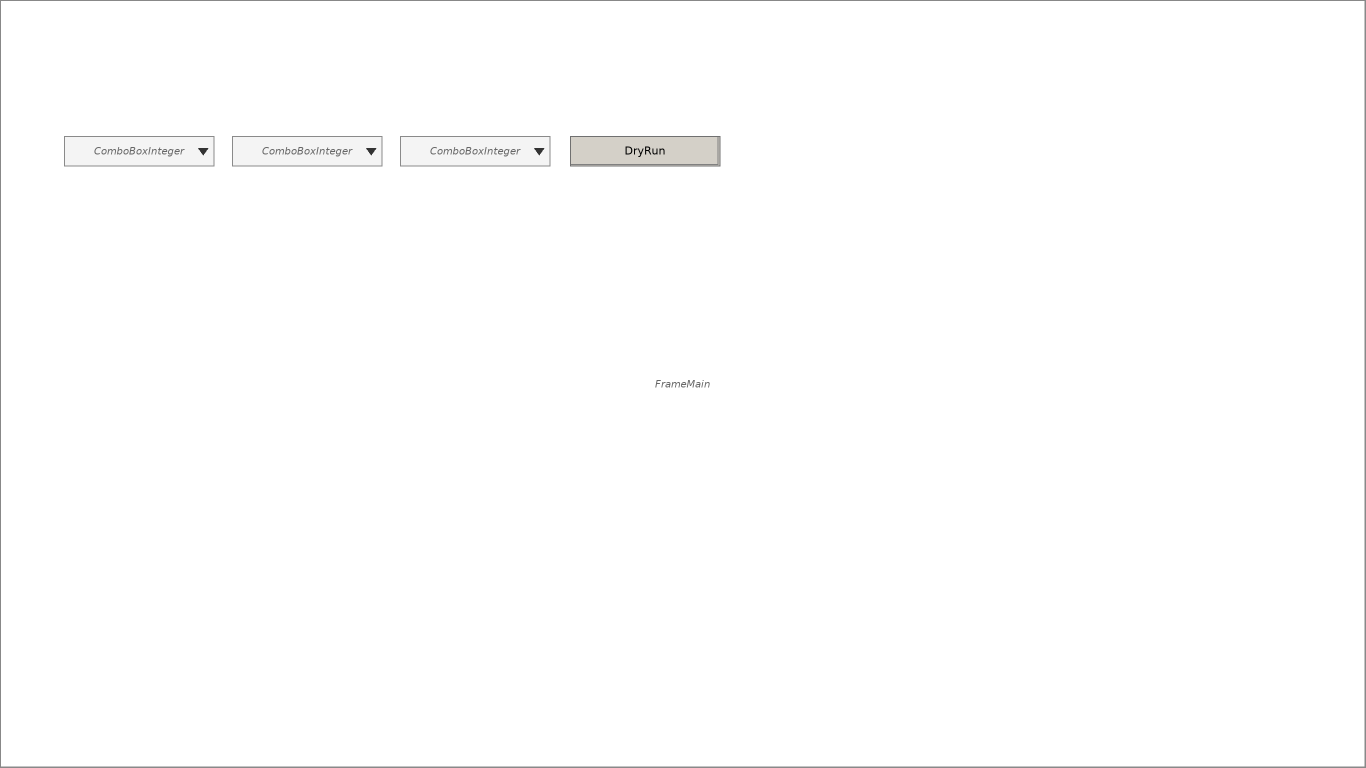
VISUALIZATION PageData  // 1366x768
    Frame (0,0 1366x768)
        shows FrameMain()
    ComboBoxInteger (64,136 150x30), variable: GVL_Data.stRecipe.eLoadClose, text list: 'LineLoadClose'
    ComboBoxInteger (232,136 150x30), variable: GVL_Data.stRecipe.eLineClose, text list: 'LineClose'
    ComboBoxInteger (400,136 150x30), variable: GVL_Data.stRecipe.eLoadPriority, text list: 'LoadPriority'
    Button (570,136 150x30), "DryRun"
        toggle GVL.stSetting.bDryRun
END_VISUALIZATION

(* stored: Version 1.1.0.1, ProductVersion 3.1.4024.3
   Visu PageData: Id {0b2b5a27-2634-4cb9-8f58-77bd32f946b4} *)
